(* CoDeSys 2.3 export: TRAFO.EXP *)

(* Data type in MNG_TCPIP *)
TYPE TRAFO :(* position and orientation as a 4x4 matrix *)
STRUCT
	baseX : VEC3; 
	fill0 : REAL;
	baseY : VEC3; 
	fill1 : REAL;
	baseZ : VEC3; 
	fill2 : REAL;
	origin : VEC3;
	fill3 : REAL;
END_STRUCT
END_TYPE
